(* CODESYS project IndraLogic.project

Project tree, tasks and I/O mapping:
  IndraMotionMlc1 : IndraMotion MLC L25, Bosch Rexroth AG, order no. R911171363, version 14.20.34.0
    application Application
      task PlcTask (cyclic, interval 10 ms, priority 5, watchdog 100 ms x 2) calls PlcProg, Datensimulator
      global variables UserVarGlobal
      Symbols
      visualisation Visualization
      global variables MlcVarGlobal
      visualisation TestFrame
      image pool ImagePool
      Funktionsbausteine/
        function block GenAngleTest [ST]
        function block GenNumTest [ST]
        function block TestGen [FBD]
      Programme/
        program PlcProg [ST]
        program Datensimulator [ST]
        program Visualisierungssteuerung [ST]
      Struktur/
        data type TestStruct
      Bedinpult_Visu/
        program PrgBedinpult_Visu [LD]
    Inline_I_O : Inline I/O, Bosch Rexroth AG, version 12.8.2.0
    Sercos_III_Master : SercosIII Master, Rexroth, order no. 1, version 14.6.0.0
  text list GlobalTextList
  5ce3da45-db07-42e7-a21c-a00fff4ed8f6|C:\Users\Kun\Desktop\Uni\Automatisierungstechnik\ProjektaufgabeAT\Overlay.png
*)

// IndraMotionMlc1/Application/Struktur/TestStruct
TYPE TestStruct :
STRUCT
	bEnable		: BOOL;
	startValue	: INT;
	finalValue	: INT;
	sweepTime	: INT;
	testActive	: BOOL := FALSE;
END_STRUCT
END_TYPE

// IndraMotionMlc1/Application/UserVarGlobal
{attribute 'qualified_only'}
VAR_GLOBAL
	testMode 		: BOOL := TRUE;
END_VAR

// IndraMotionMlc1/Application/MlcVarGlobal
(* Automatically generated code by XLC/MLC. *)
(* Please don't edit, the code will be overwritten. For usercode use UserVarGlobal! *)
{attribute 'linkalways'}
{attribute 'analysis' := '-33'}
VAR_GLOBAL CONSTANT

(*Probe 001*)
TouchProbe001: TOUCHPROBE_REF :=(CntrlNo:=LOCAL_CNTRL,TouchProbeNo:=TOUCHPROBE_1);

(*Probe 002*)
TouchProbe002: TOUCHPROBE_REF :=(CntrlNo:=LOCAL_CNTRL,TouchProbeNo:=TOUCHPROBE_2);

(*Probe 003*)
TouchProbe003: TOUCHPROBE_REF :=(CntrlNo:=LOCAL_CNTRL,TouchProbeNo:=TOUCHPROBE_3);

(*Probe 004*)
TouchProbe004: TOUCHPROBE_REF :=(CntrlNo:=LOCAL_CNTRL,TouchProbeNo:=TOUCHPROBE_4);

(*Probe 005*)
TouchProbe005: TOUCHPROBE_REF :=(CntrlNo:=LOCAL_CNTRL,TouchProbeNo:=TOUCHPROBE_5);

(*Probe 006*)
TouchProbe006: TOUCHPROBE_REF :=(CntrlNo:=LOCAL_CNTRL,TouchProbeNo:=TOUCHPROBE_6);

(*Probe 007*)
TouchProbe007: TOUCHPROBE_REF :=(CntrlNo:=LOCAL_CNTRL,TouchProbeNo:=TOUCHPROBE_7);

(*Probe 008*)
TouchProbe008: TOUCHPROBE_REF :=(CntrlNo:=LOCAL_CNTRL,TouchProbeNo:=TOUCHPROBE_8);

(*Probe 009*)
TouchProbe009: TOUCHPROBE_REF :=(CntrlNo:=LOCAL_CNTRL,TouchProbeNo:=TOUCHPROBE_9);

(*Probe 010*)
TouchProbe010: TOUCHPROBE_REF :=(CntrlNo:=LOCAL_CNTRL,TouchProbeNo:=TOUCHPROBE_10);

(*Probe 011*)
TouchProbe011: TOUCHPROBE_REF :=(CntrlNo:=LOCAL_CNTRL,TouchProbeNo:=TOUCHPROBE_11);

(*Probe 012*)
TouchProbe012: TOUCHPROBE_REF :=(CntrlNo:=LOCAL_CNTRL,TouchProbeNo:=TOUCHPROBE_12);

(*Probe 013*)
TouchProbe013: TOUCHPROBE_REF :=(CntrlNo:=LOCAL_CNTRL,TouchProbeNo:=TOUCHPROBE_13);

(*Probe 014*)
TouchProbe014: TOUCHPROBE_REF :=(CntrlNo:=LOCAL_CNTRL,TouchProbeNo:=TOUCHPROBE_14);

(*Probe 015*)
TouchProbe015: TOUCHPROBE_REF :=(CntrlNo:=LOCAL_CNTRL,TouchProbeNo:=TOUCHPROBE_15);

(*Probe 016*)
TouchProbe016: TOUCHPROBE_REF :=(CntrlNo:=LOCAL_CNTRL,TouchProbeNo:=TOUCHPROBE_16);

(*Probe 017*)
TouchProbe017: TOUCHPROBE_REF :=(CntrlNo:=LOCAL_CNTRL,TouchProbeNo:=TOUCHPROBE_17);

(*Probe 018*)
TouchProbe018: TOUCHPROBE_REF :=(CntrlNo:=LOCAL_CNTRL,TouchProbeNo:=TOUCHPROBE_18);

(*Probe 019*)
TouchProbe019: TOUCHPROBE_REF :=(CntrlNo:=LOCAL_CNTRL,TouchProbeNo:=TOUCHPROBE_19);

(*Probe 020*)
TouchProbe020: TOUCHPROBE_REF :=(CntrlNo:=LOCAL_CNTRL,TouchProbeNo:=TOUCHPROBE_20);

(*Probe 021*)
TouchProbe021: TOUCHPROBE_REF :=(CntrlNo:=LOCAL_CNTRL,TouchProbeNo:=TOUCHPROBE_21);

(*Probe 022*)
TouchProbe022: TOUCHPROBE_REF :=(CntrlNo:=LOCAL_CNTRL,TouchProbeNo:=TOUCHPROBE_22);

(*Probe 023*)
TouchProbe023: TOUCHPROBE_REF :=(CntrlNo:=LOCAL_CNTRL,TouchProbeNo:=TOUCHPROBE_23);

(*Probe 024*)
TouchProbe024: TOUCHPROBE_REF :=(CntrlNo:=LOCAL_CNTRL,TouchProbeNo:=TOUCHPROBE_24);

(*Probe 025*)
TouchProbe025: TOUCHPROBE_REF :=(CntrlNo:=LOCAL_CNTRL,TouchProbeNo:=TOUCHPROBE_25);

(*Probe 026*)
TouchProbe026: TOUCHPROBE_REF :=(CntrlNo:=LOCAL_CNTRL,TouchProbeNo:=TOUCHPROBE_26);

(*Probe 027*)
TouchProbe027: TOUCHPROBE_REF :=(CntrlNo:=LOCAL_CNTRL,TouchProbeNo:=TOUCHPROBE_27);

(*Probe 028*)
TouchProbe028: TOUCHPROBE_REF :=(CntrlNo:=LOCAL_CNTRL,TouchProbeNo:=TOUCHPROBE_28);

(*Probe 029*)
TouchProbe029: TOUCHPROBE_REF :=(CntrlNo:=LOCAL_CNTRL,TouchProbeNo:=TOUCHPROBE_29);

(*Probe 030*)
TouchProbe030: TOUCHPROBE_REF :=(CntrlNo:=LOCAL_CNTRL,TouchProbeNo:=TOUCHPROBE_30);

(*Probe 031*)
TouchProbe031: TOUCHPROBE_REF :=(CntrlNo:=LOCAL_CNTRL,TouchProbeNo:=TOUCHPROBE_31);

(*Probe 032*)
TouchProbe032: TOUCHPROBE_REF :=(CntrlNo:=LOCAL_CNTRL,TouchProbeNo:=TOUCHPROBE_32);

(*Probe 033*)
TouchProbe033: TOUCHPROBE_REF :=(CntrlNo:=LOCAL_CNTRL,TouchProbeNo:=TOUCHPROBE_33);

(*Probe 034*)
TouchProbe034: TOUCHPROBE_REF :=(CntrlNo:=LOCAL_CNTRL,TouchProbeNo:=TOUCHPROBE_34);

(*Probe 035*)
TouchProbe035: TOUCHPROBE_REF :=(CntrlNo:=LOCAL_CNTRL,TouchProbeNo:=TOUCHPROBE_35);

(*Probe 036*)
TouchProbe036: TOUCHPROBE_REF :=(CntrlNo:=LOCAL_CNTRL,TouchProbeNo:=TOUCHPROBE_36);

(*Probe 037*)
TouchProbe037: TOUCHPROBE_REF :=(CntrlNo:=LOCAL_CNTRL,TouchProbeNo:=TOUCHPROBE_37);

(*Probe 038*)
TouchProbe038: TOUCHPROBE_REF :=(CntrlNo:=LOCAL_CNTRL,TouchProbeNo:=TOUCHPROBE_38);

(*Probe 039*)
TouchProbe039: TOUCHPROBE_REF :=(CntrlNo:=LOCAL_CNTRL,TouchProbeNo:=TOUCHPROBE_39);

(*Probe 040*)
TouchProbe040: TOUCHPROBE_REF :=(CntrlNo:=LOCAL_CNTRL,TouchProbeNo:=TOUCHPROBE_40);

(*Probe 041*)
TouchProbe041: TOUCHPROBE_REF :=(CntrlNo:=LOCAL_CNTRL,TouchProbeNo:=TOUCHPROBE_41);

(*Probe 042*)
TouchProbe042: TOUCHPROBE_REF :=(CntrlNo:=LOCAL_CNTRL,TouchProbeNo:=TOUCHPROBE_42);

(*Probe 043*)
TouchProbe043: TOUCHPROBE_REF :=(CntrlNo:=LOCAL_CNTRL,TouchProbeNo:=TOUCHPROBE_43);

(*Probe 044*)
TouchProbe044: TOUCHPROBE_REF :=(CntrlNo:=LOCAL_CNTRL,TouchProbeNo:=TOUCHPROBE_44);

(*Probe 045*)
TouchProbe045: TOUCHPROBE_REF :=(CntrlNo:=LOCAL_CNTRL,TouchProbeNo:=TOUCHPROBE_45);

(*Probe 046*)
TouchProbe046: TOUCHPROBE_REF :=(CntrlNo:=LOCAL_CNTRL,TouchProbeNo:=TOUCHPROBE_46);

(*Probe 047*)
TouchProbe047: TOUCHPROBE_REF :=(CntrlNo:=LOCAL_CNTRL,TouchProbeNo:=TOUCHPROBE_47);

(*Probe 048*)
TouchProbe048: TOUCHPROBE_REF :=(CntrlNo:=LOCAL_CNTRL,TouchProbeNo:=TOUCHPROBE_48);

(*Probe 049*)
TouchProbe049: TOUCHPROBE_REF :=(CntrlNo:=LOCAL_CNTRL,TouchProbeNo:=TOUCHPROBE_49);

(*Probe 050*)
TouchProbe050: TOUCHPROBE_REF :=(CntrlNo:=LOCAL_CNTRL,TouchProbeNo:=TOUCHPROBE_50);

(*Probe 051*)
TouchProbe051: TOUCHPROBE_REF :=(CntrlNo:=LOCAL_CNTRL,TouchProbeNo:=TOUCHPROBE_51);

(*Probe 052*)
TouchProbe052: TOUCHPROBE_REF :=(CntrlNo:=LOCAL_CNTRL,TouchProbeNo:=TOUCHPROBE_52);

(*Probe 053*)
TouchProbe053: TOUCHPROBE_REF :=(CntrlNo:=LOCAL_CNTRL,TouchProbeNo:=TOUCHPROBE_53);

(*Probe 054*)
TouchProbe054: TOUCHPROBE_REF :=(CntrlNo:=LOCAL_CNTRL,TouchProbeNo:=TOUCHPROBE_54);

(*Probe 055*)
TouchProbe055: TOUCHPROBE_REF :=(CntrlNo:=LOCAL_CNTRL,TouchProbeNo:=TOUCHPROBE_55);

(*Probe 056*)
TouchProbe056: TOUCHPROBE_REF :=(CntrlNo:=LOCAL_CNTRL,TouchProbeNo:=TOUCHPROBE_56);

(*Probe 057*)
TouchProbe057: TOUCHPROBE_REF :=(CntrlNo:=LOCAL_CNTRL,TouchProbeNo:=TOUCHPROBE_57);

(*Probe 058*)
TouchProbe058: TOUCHPROBE_REF :=(CntrlNo:=LOCAL_CNTRL,TouchProbeNo:=TOUCHPROBE_58);

(*Probe 059*)
TouchProbe059: TOUCHPROBE_REF :=(CntrlNo:=LOCAL_CNTRL,TouchProbeNo:=TOUCHPROBE_59);

(*Probe 060*)
TouchProbe060: TOUCHPROBE_REF :=(CntrlNo:=LOCAL_CNTRL,TouchProbeNo:=TOUCHPROBE_60);

(*Probe 061*)
TouchProbe061: TOUCHPROBE_REF :=(CntrlNo:=LOCAL_CNTRL,TouchProbeNo:=TOUCHPROBE_61);

(*Probe 062*)
TouchProbe062: TOUCHPROBE_REF :=(CntrlNo:=LOCAL_CNTRL,TouchProbeNo:=TOUCHPROBE_62);

(*Probe 063*)
TouchProbe063: TOUCHPROBE_REF :=(CntrlNo:=LOCAL_CNTRL,TouchProbeNo:=TOUCHPROBE_63);

(*Probe 064*)
TouchProbe064: TOUCHPROBE_REF :=(CntrlNo:=LOCAL_CNTRL,TouchProbeNo:=TOUCHPROBE_64);

(*Probe 065*)
TouchProbe065: TOUCHPROBE_REF :=(CntrlNo:=LOCAL_CNTRL,TouchProbeNo:=TOUCHPROBE_65);

(*Probe 066*)
TouchProbe066: TOUCHPROBE_REF :=(CntrlNo:=LOCAL_CNTRL,TouchProbeNo:=TOUCHPROBE_66);

(*Probe 067*)
TouchProbe067: TOUCHPROBE_REF :=(CntrlNo:=LOCAL_CNTRL,TouchProbeNo:=TOUCHPROBE_67);

(*Probe 068*)
TouchProbe068: TOUCHPROBE_REF :=(CntrlNo:=LOCAL_CNTRL,TouchProbeNo:=TOUCHPROBE_68);

(*Probe 069*)
TouchProbe069: TOUCHPROBE_REF :=(CntrlNo:=LOCAL_CNTRL,TouchProbeNo:=TOUCHPROBE_69);

(*Probe 070*)
TouchProbe070: TOUCHPROBE_REF :=(CntrlNo:=LOCAL_CNTRL,TouchProbeNo:=TOUCHPROBE_70);

(*Probe 071*)
TouchProbe071: TOUCHPROBE_REF :=(CntrlNo:=LOCAL_CNTRL,TouchProbeNo:=TOUCHPROBE_71);

(*Probe 072*)
TouchProbe072: TOUCHPROBE_REF :=(CntrlNo:=LOCAL_CNTRL,TouchProbeNo:=TOUCHPROBE_72);

(*Probe 073*)
TouchProbe073: TOUCHPROBE_REF :=(CntrlNo:=LOCAL_CNTRL,TouchProbeNo:=TOUCHPROBE_73);

(*Probe 074*)
TouchProbe074: TOUCHPROBE_REF :=(CntrlNo:=LOCAL_CNTRL,TouchProbeNo:=TOUCHPROBE_74);

(*Probe 075*)
TouchProbe075: TOUCHPROBE_REF :=(CntrlNo:=LOCAL_CNTRL,TouchProbeNo:=TOUCHPROBE_75);

(*Probe 076*)
TouchProbe076: TOUCHPROBE_REF :=(CntrlNo:=LOCAL_CNTRL,TouchProbeNo:=TOUCHPROBE_76);

(*Probe 077*)
TouchProbe077: TOUCHPROBE_REF :=(CntrlNo:=LOCAL_CNTRL,TouchProbeNo:=TOUCHPROBE_77);

(*Probe 078*)
TouchProbe078: TOUCHPROBE_REF :=(CntrlNo:=LOCAL_CNTRL,TouchProbeNo:=TOUCHPROBE_78);

(*Probe 079*)
TouchProbe079: TOUCHPROBE_REF :=(CntrlNo:=LOCAL_CNTRL,TouchProbeNo:=TOUCHPROBE_79);

(*Probe 080*)
TouchProbe080: TOUCHPROBE_REF :=(CntrlNo:=LOCAL_CNTRL,TouchProbeNo:=TOUCHPROBE_80);

(*Probe 081*)
TouchProbe081: TOUCHPROBE_REF :=(CntrlNo:=LOCAL_CNTRL,TouchProbeNo:=TOUCHPROBE_81);

(*Probe 082*)
TouchProbe082: TOUCHPROBE_REF :=(CntrlNo:=LOCAL_CNTRL,TouchProbeNo:=TOUCHPROBE_82);

(*Probe 083*)
TouchProbe083: TOUCHPROBE_REF :=(CntrlNo:=LOCAL_CNTRL,TouchProbeNo:=TOUCHPROBE_83);

(*Probe 084*)
TouchProbe084: TOUCHPROBE_REF :=(CntrlNo:=LOCAL_CNTRL,TouchProbeNo:=TOUCHPROBE_84);

(*Probe 085*)
TouchProbe085: TOUCHPROBE_REF :=(CntrlNo:=LOCAL_CNTRL,TouchProbeNo:=TOUCHPROBE_85);

(*Probe 086*)
TouchProbe086: TOUCHPROBE_REF :=(CntrlNo:=LOCAL_CNTRL,TouchProbeNo:=TOUCHPROBE_86);

(*Probe 087*)
TouchProbe087: TOUCHPROBE_REF :=(CntrlNo:=LOCAL_CNTRL,TouchProbeNo:=TOUCHPROBE_87);

(*Probe 088*)
TouchProbe088: TOUCHPROBE_REF :=(CntrlNo:=LOCAL_CNTRL,TouchProbeNo:=TOUCHPROBE_88);

(*Probe 089*)
TouchProbe089: TOUCHPROBE_REF :=(CntrlNo:=LOCAL_CNTRL,TouchProbeNo:=TOUCHPROBE_89);

(*Probe 090*)
TouchProbe090: TOUCHPROBE_REF :=(CntrlNo:=LOCAL_CNTRL,TouchProbeNo:=TOUCHPROBE_90);

(*Probe 091*)
TouchProbe091: TOUCHPROBE_REF :=(CntrlNo:=LOCAL_CNTRL,TouchProbeNo:=TOUCHPROBE_91);

(*Probe 092*)
TouchProbe092: TOUCHPROBE_REF :=(CntrlNo:=LOCAL_CNTRL,TouchProbeNo:=TOUCHPROBE_92);

(*Probe 093*)
TouchProbe093: TOUCHPROBE_REF :=(CntrlNo:=LOCAL_CNTRL,TouchProbeNo:=TOUCHPROBE_93);

(*Probe 094*)
TouchProbe094: TOUCHPROBE_REF :=(CntrlNo:=LOCAL_CNTRL,TouchProbeNo:=TOUCHPROBE_94);

(*Probe 095*)
TouchProbe095: TOUCHPROBE_REF :=(CntrlNo:=LOCAL_CNTRL,TouchProbeNo:=TOUCHPROBE_95);

(*Probe 096*)
TouchProbe096: TOUCHPROBE_REF :=(CntrlNo:=LOCAL_CNTRL,TouchProbeNo:=TOUCHPROBE_96);

(*Probe 097*)
TouchProbe097: TOUCHPROBE_REF :=(CntrlNo:=LOCAL_CNTRL,TouchProbeNo:=TOUCHPROBE_97);

(*Probe 098*)
TouchProbe098: TOUCHPROBE_REF :=(CntrlNo:=LOCAL_CNTRL,TouchProbeNo:=TOUCHPROBE_98);

(*Probe 099*)
TouchProbe099: TOUCHPROBE_REF :=(CntrlNo:=LOCAL_CNTRL,TouchProbeNo:=TOUCHPROBE_99);

(*Probe 100*)
TouchProbe100: TOUCHPROBE_REF :=(CntrlNo:=LOCAL_CNTRL,TouchProbeNo:=TOUCHPROBE_100);

END_VAR

// IndraMotionMlc1/Application/Programme/PlcProg
PROGRAM PlcProg
VAR
	rPitch 		: 	SINT;
	rRoll 		: 	REAL;
	height		:	INT;
	speed		:	UINT	:=	10;
	climbRate	:	REAL;
	Direction	:	INT;
	steps		:	LINT;
	bEnableTest	:	BOOL 	:= FALSE;
	rollTest	:	GenAngleTest;
	heightTest	:	GenNumTest;
	testGenerator	:	TestGen;
	rollTestStruct	:	testStruct;
	heightTestStruct:	testStruct;
END_VAR

VAR CONSTANT
	timestep	:	INT		:=	5;	// Timestep
	
END_VAR

(* 
rollTest(benable:=bEnableTest,startAngle:=-20.0,finalAngle:=20.0,sweepTime:=500);
rRoll := rollTest.Angle/1;
IF (rollTest.active = FALSE) THEN
	rRoll := 0;
END_IF
*)
(*
rollTestStruct.bEnable 		:= bEnableTest;
rollTestStruct.startValue 	:= -20;
rollTestStruct.finalValue 	:= 20;
rollTestStruct.sweepTime 	:= 500;
testGenerator(rollTestStruct := rollTestStruct);
rRoll := testGenerator.roll;
heightTest(benable:=bEnableTest,startNum:=0,finalNum:=4000,sweepTime:=500);
height := heightTest.num;
*)

rRoll := Datensimulator.rRoll;
height := Datensimulator.height;

END_PROGRAM

// IndraMotionMlc1/Application/Programme/Datensimulator
PROGRAM Datensimulator
VAR
	testMode		:	BOOL;
	rPitch 			: 	REAL;
	rRoll 			: 	REAL;
	height			:	INT;
	speed			:	UINT;
	climbRate		:	REAL;
	Direction		:	REAL;
	steps			:	LINT;
	testGenerator	:	TestGen;
	rollTestStruct	:	testStruct;
	heightTestStruct:	testStruct;
	test			: BOOL;
END_VAR

IF (UserVarGlobal.testMode) THEN
	rollTestStruct.bEnable 		:= TRUE;
	rollTestStruct.startValue 	:= -20;
	rollTestStruct.finalValue 	:= 20;
	rollTestStruct.sweepTime 	:= 500;
	
	heightTestStruct.bEnable 	:= TRUE;
	heightTestStruct.startValue	:= 0;
	heightTestStruct.finalValue := 2000;
	heightTestStruct.sweepTime	:= 300;
	
	testGenerator(rollTestStruct:=rollTestStruct , heightTestStruct:=heightTestStruct);
	
	rRoll := testGenerator.roll;
	height := testGenerator.height;
	test :=  testGenerator.testActive;
END_IF

END_PROGRAM

// IndraMotionMlc1/Application/Funktionsbausteine/TestGen
FUNCTION_BLOCK TestGen
VAR_INPUT
	pitchTestStruct		: TestStruct;
	rollTestStruct		: TestStruct;
	heightTestStruct	: TestStruct;
	speedTestStruct		: TestStruct;
	climbRateTestStruct	: TestStruct;
	directionTestStruct	: TestStruct;
END_VAR
VAR_OUTPUT
	pitch			: REAL;
	roll			: REAL;
	height			: INT;
	speed			: UINT;
	climbRate		: REAL;
	direction		: REAL;
	testActive		: BOOL;
END_VAR
VAR
	pitchTest		: GenAngleTest;
	rollTest		: GenAngleTest;
	heightTest		: GenNumTest;
	speedTest		: GenNumTest;
	climbRateTest	: GenNumTest;
	directionTest	: GenAngleTest;
END_VAR

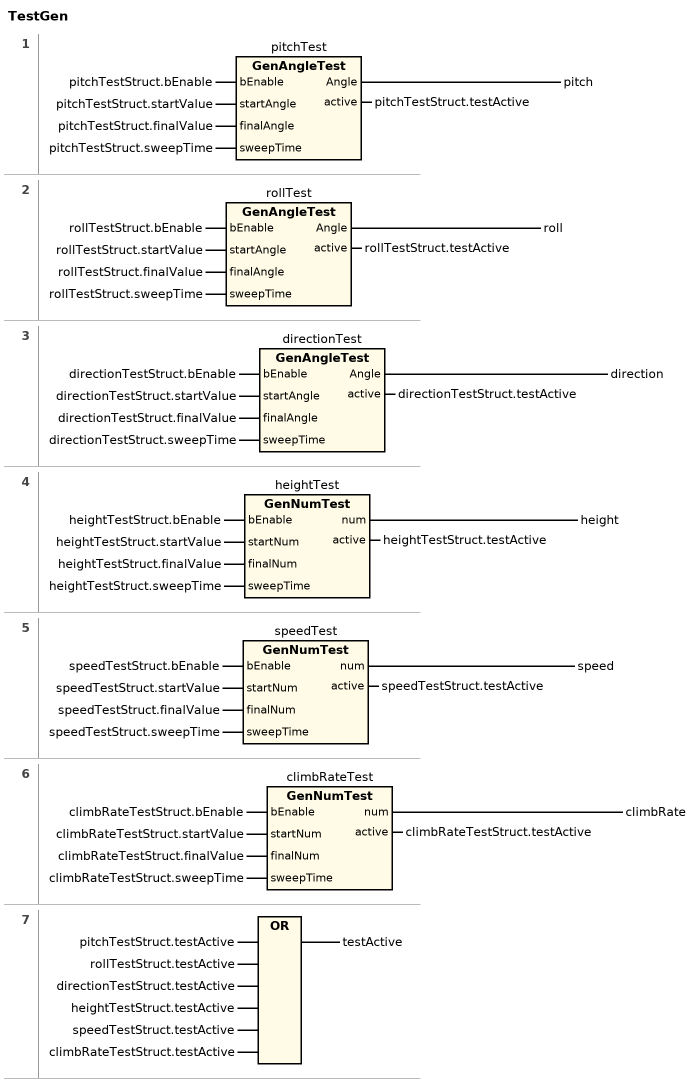
// NETWORK 1
pitchTest(
    bEnable := pitchTestStruct.bEnable,
    startAngle := pitchTestStruct.startValue,
    finalAngle := pitchTestStruct.finalValue,
    sweepTime := pitchTestStruct.sweepTime,
    active => pitchTestStruct.testActive); // GenAngleTest
pitch := pitchTest.Angle;

// NETWORK 2
rollTest(
    bEnable := rollTestStruct.bEnable,
    startAngle := rollTestStruct.startValue,
    finalAngle := rollTestStruct.finalValue,
    sweepTime := rollTestStruct.sweepTime,
    active => rollTestStruct.testActive); // GenAngleTest
roll := rollTest.Angle;

// NETWORK 3
directionTest(
    bEnable := directionTestStruct.bEnable,
    startAngle := directionTestStruct.startValue,
    finalAngle := directionTestStruct.finalValue,
    sweepTime := directionTestStruct.sweepTime,
    active => directionTestStruct.testActive); // GenAngleTest
direction := directionTest.Angle;

// NETWORK 4
heightTest(
    bEnable := heightTestStruct.bEnable,
    startNum := heightTestStruct.startValue,
    finalNum := heightTestStruct.finalValue,
    sweepTime := heightTestStruct.sweepTime,
    active => heightTestStruct.testActive); // GenNumTest
height := heightTest.num;

// NETWORK 5
speedTest(
    bEnable := speedTestStruct.bEnable,
    startNum := speedTestStruct.startValue,
    finalNum := speedTestStruct.finalValue,
    sweepTime := speedTestStruct.sweepTime,
    active => speedTestStruct.testActive); // GenNumTest
speed := speedTest.num;

// NETWORK 6
climbRateTest(
    bEnable := climbRateTestStruct.bEnable,
    startNum := climbRateTestStruct.startValue,
    finalNum := climbRateTestStruct.finalValue,
    sweepTime := climbRateTestStruct.sweepTime,
    active => climbRateTestStruct.testActive); // GenNumTest
climbRate := climbRateTest.num;

// NETWORK 7
testActive := pitchTestStruct.testActive OR rollTestStruct.testActive OR directionTestStruct.testActive OR heightTestStruct.testActive OR speedTestStruct.testActive OR climbRateTestStruct.testActive;

END_FUNCTION_BLOCK

// IndraMotionMlc1/Application/Funktionsbausteine/GenAngleTest
FUNCTION_BLOCK GenAngleTest
VAR_INPUT
	bEnable			: BOOL;
	startAngle		: REAL;
	finalAngle		: REAL;
	sweepTime		: INT;	//Sweeptime in cycles
END_VAR
VAR_OUTPUT
	Angle			: REAL;
	active			: BOOL;
END_VAR
VAR
	internalTimer	: INT;
	angleInc		: REAL;
	bFirstSweep		: BOOL := TRUE;	// Winkel soll einmal in beide Richtugnen veränder werden
END_VAR

angleInc := -(startAngle-finalAngle)/sweepTime;
IF (bEnable AND internalTimer < sweepTime AND bFirstSweep) THEN
	Angle := startAngle + angleInc * internalTimer;
	internalTimer := internalTimer + 1;
	active := TRUE;
ELSIF (internalTimer = sweepTime) THEN
	bFirstSweep := FALSE;
END_IF
IF (bFirstSweep = FALSE AND internalTimer > 0) THEN
	Angle := finalAngle + angleInc * (internalTimer-sweepTime);
	internalTimer := internalTimer - 1;
ELSIF (bFirstSweep = FALSE AND internalTimer = 0) THEN
	active := FALSE;
END_IF
IF (bEnable = FALSE) THEN
	Angle := 0;
	internalTimer := 0;
	angleInc := 0;
	bFirstSweep := TRUE;
	active := FALSE;
END_IF

END_FUNCTION_BLOCK

// IndraMotionMlc1/Application/Funktionsbausteine/GenNumTest
FUNCTION_BLOCK GenNumTest
VAR_INPUT
	bEnable			: BOOL;
	startNum		: INT;
	finalNum		: INT;
	sweepTime		: INT;	//Sweeptime in cycles
END_VAR
VAR_OUTPUT
	num				: INT;
	active			: BOOL;
END_VAR
VAR
	internalTimer	: INT;
	inc				: INT;
	bFirstSweep		: BOOL	:= TRUE;
END_VAR

IF bEnable THEN
	inc := -(startNum-finalNum)/sweepTime;
END_IF
IF (bEnable AND internalTimer < sweepTime AND bFirstSweep) THEN
	num := startNum + inc * internalTimer;
	internalTimer := internalTimer + 1;
	active := TRUE;
ELSIF (internalTimer = sweepTime) THEN
	bFirstSweep := FALSE;
	num := finalNum;
END_IF
IF (bFirstSweep = FALSE AND internalTimer > 0) THEN
	num := finalNum + inc * (internalTimer-sweepTime);
	internalTimer := internalTimer - 1;
ELSIF (bFirstSweep = FALSE AND internalTimer = 0) THEN
	active := FALSE;
	num := startNum;
END_IF
IF (bEnable = FALSE) THEN
	num := 0;
	internalTimer := 0;
	inc := 0;
	bFirstSweep := TRUE;
	active := FALSE;
END_IF

END_FUNCTION_BLOCK

// IndraMotionMlc1/Application/Programme/Visualisierungssteuerung
PROGRAM Visualisierungssteuerung
VAR
END_VAR

END_PROGRAM

// IndraMotionMlc1/Application/Bedinpult_Visu/PrgBedinpult_Visu
PROGRAM PrgBedinpult_Visu
VAR
bTaster_AUS_Visu 					: BOOL; // Anlage Aus - Achtung Öffner
bTaster_EIN_Visu 				 	: BOOL; // Anlage Ein 
bSchalter_Automatik_Visu		 	: BOOL; // Umschalter Automatik =1 / Handbetrieb =0 
END_VAR

// NETWORK 1

END_PROGRAM

// IndraMotionMlc1/Application/Visualization
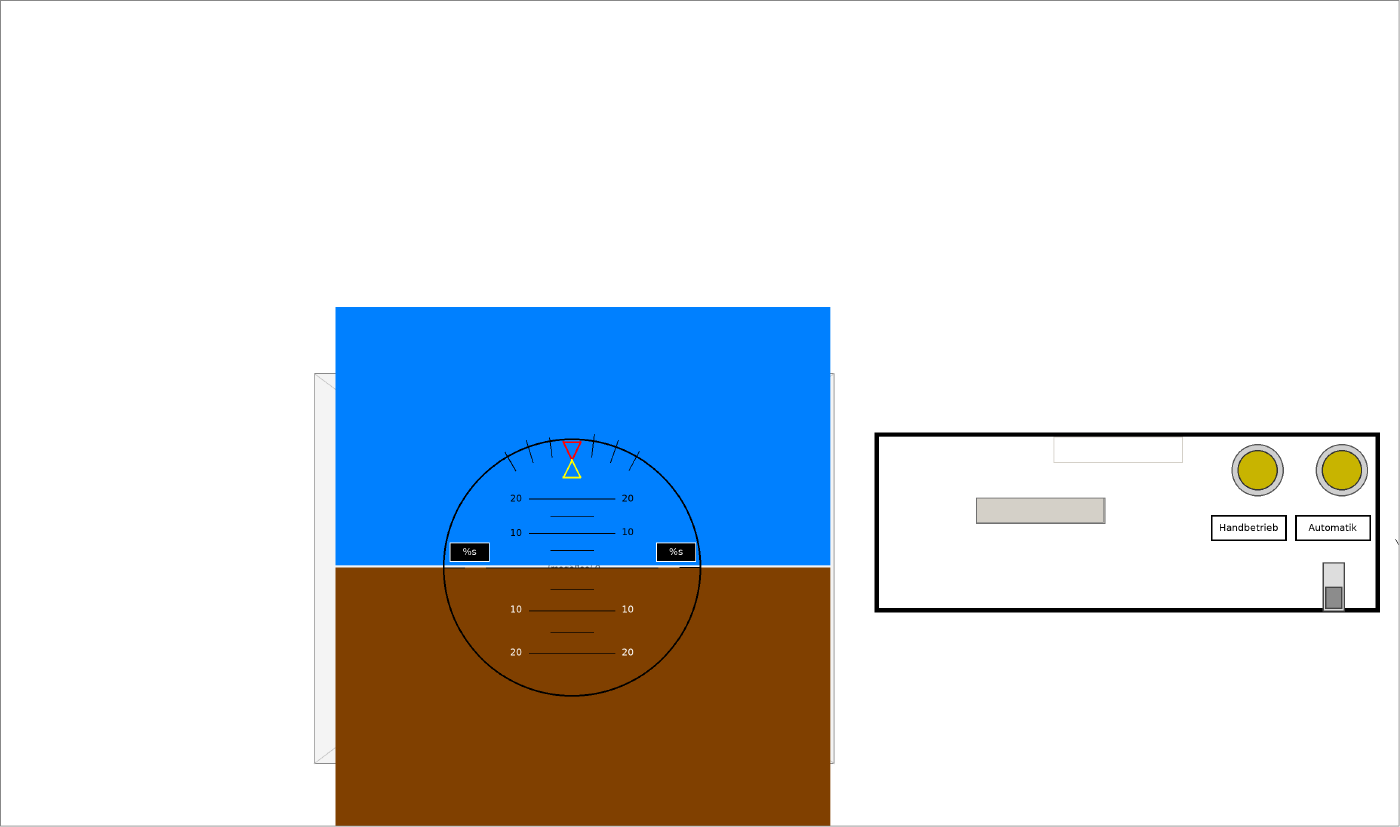
VISUALIZATION Visualization  // 1628x962
    Image (365,434 605x454), image: ImagePool.0
    Rectangle (390,660 575x300)
        p2858320360: PlcProg.rRoll
        p2773130477: PlcProg.rPitch
        p1126004900: PlcProg.rPitch
    Rectangle (390,357 575x300)
        p2858320360: PlcProg.rRoll
        p2773130477: PlcProg.rPitch
        p1126004900: PlcProg.rPitch
    Ellipse (515,510 300x300)
    Line (565,660) (765,660)
    Line (640,640) (690,640)
        p2858320360: PlcProg.rRoll
        p2773130477: PlcProg.rPitch
        p1126004900: PlcProg.rPitch
    Line (615,620) (715,620)
        p2858320360: PlcProg.rRoll
        p2773130477: PlcProg.rPitch
        p1126004900: PlcProg.rPitch
    Line (640,600) (690,600)
        p2858320360: PlcProg.rRoll
        p2773130477: PlcProg.rPitch
        p1126004900: PlcProg.rPitch
    Line (640,685) (690,685)
        p2858320360: PlcProg.rRoll
        p2773130477: PlcProg.rPitch
        p1126004900: PlcProg.rPitch
    Line (615,710) (715,710)
        p2858320360: PlcProg.rRoll
        p2773130477: PlcProg.rPitch
        p1126004900: PlcProg.rPitch
    Line (640,735) (690,735)
        p2858320360: PlcProg.rRoll
        p2773130477: PlcProg.rPitch
        p1126004900: PlcProg.rPitch
    Line (615,580) (715,580)
        p2858320360: PlcProg.rRoll
        p2773130477: PlcProg.rPitch
        p1126004900: PlcProg.rPitch
    Line (615,760) (715,760)
        p2858320360: PlcProg.rRoll
        p2773130477: PlcProg.rPitch
        p1126004900: PlcProg.rPitch
    Line (815,660) (790,660)
    Line (515,660) (540,660)
    Rectangle (715,605 30x28), "10"
        p2858320360: PlcProg.rRoll
        p2773130477: PlcProg.rPitch
        p1126004900: PlcProg.rPitch
    Rectangle (715,565 30x30), "20"
        p2858320360: PlcProg.rRoll
        p2773130477: PlcProg.rPitch
        p1126004900: PlcProg.rPitch
    Rectangle (585,605 30x30), "10"
        p2858320360: PlcProg.rRoll
        p2773130477: PlcProg.rPitch
        p1126004900: PlcProg.rPitch
    Rectangle (585,565 30x30), "20"
        p2858320360: PlcProg.rRoll
        p2773130477: PlcProg.rPitch
        p1126004900: PlcProg.rPitch
    Polyline (655,514) (655,514) (675,514) (665,535) (655,514)
    Rectangle (715,695 30x28), "10"
        p2858320360: PlcProg.rRoll
        p2773130477: PlcProg.rPitch
        p1126004900: PlcProg.rPitch
    Rectangle (585,695 30x28), "10"
        p2858320360: PlcProg.rRoll
        p2773130477: PlcProg.rPitch
        p1126004900: PlcProg.rPitch
    Rectangle (715,745 30x28), "20"
        p2858320360: PlcProg.rRoll
        p2773130477: PlcProg.rPitch
        p1126004900: PlcProg.rPitch
    Rectangle (585,745 30x28), "20"
        p2858320360: PlcProg.rRoll
    Polyline (654,555) (655,555) (675,555) (665,535) (655,555)
        p2858320360: PlcProg.rRoll
    RoundedRectangle (763,631 46x22), "%s", text variable: PlcProg.height, text index: PlcProg.speed
    RoundedRectangle (523,631 46x22), "%s", text variable: PlcProg.speed
    Line (743,525) (731,547)
    Line (710,538) (719,512)
    Line (688,532) (691,505)
    Line (642,532) (639,509)
    Line (620,538) (612,512)
    Line (600,548) (587,526)
    Rectangle (1017,503 587x209)
    Line (1626,633) (1623,627)
    DipSwitch (1517,654 68x57), variable: PrgBedinpult_Visu.bSchalter_Automatik_Visu, behaviour: TOGGLE, style: Switch-DipSwitch-Gray
    Lamp1 (1518,512 85x70), style: Lamp-Lamp1-Yellow
    Lamp1 (1420,512 85x70), style: Lamp-Lamp1-Yellow
    Rectangle (1506,599 88x30), "Automatik"
    Rectangle (1408,599 88x30), "Handbetrieb"
    Textfield (1225,508 150x30), input disabled if: PlcProg.bEnableTest
    Button (1135,579 150x30)
        tap PlcProg.bEnableTest
END_VISUALIZATION

// IndraMotionMlc1/Application/TestFrame
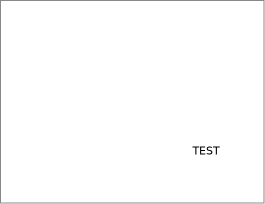
VISUALIZATION TestFrame  // 265x204
    Label (149,100 114x102), "TEST"
END_VISUALIZATION
